FUNCTION_BLOCK StartMovementsTask EXTENDS TcoMitsubishiRoboticsTask
VAR
    _moveParams : TcoAbstractions.TcoRoboticsMovementsParams;
END_VAR

IF Execute() THEN
    IF _progress = 0 THEN
        IF NOT __ISVALIDREF(inoControl) THEN
            _varInfo := __VARINFO(inoControl);
            Messenger.Programming(_sb.Clear().Append('<#Invalid reference: #>').Append(_varInfo.Symbol).ToString()).Pin();
        ELSIF NOT __ISVALIDREF(inoConfig) THEN
            _varInfo := __VARINFO(inoConfig);
            Messenger.Programming(_sb.Clear().Append('<#Invalid reference: #>').Append(_varInfo.Symbol).ToString()).Pin();
        ELSIF NOT __ISVALIDREF(inoStatus) THEN
            _varInfo := __VARINFO(inoStatus);
            Messenger.Programming(_sb.Clear().Append('<#Invalid reference: #>').Append(_varInfo.Symbol).ToString()).Pin();
        ELSE
            _progress := _progress + 1;
        END_IF
    END_IF

    IF _progress = 1 THEN
        _varInfo := __VARINFO(inoStatus.State.OperationEnable);

        THIS^.Messenger.OnCondition(_infoTimer.Q AND NOT inoStatus.State.OperationEnable)
            .Warning(_sb.Clear().Append('<#Waiting for Operation enable! #>').Append(_varInfo.Symbol).ToString());

        _varInfo := __VARINFO(inoStatus.State.AutoEnable);

        THIS^.Messenger.OnCondition(_infoTimer.Q AND NOT inoStatus.State.AutoEnable)
            .Warning(_sb.Clear().Append('<#Waiting for auto enable! #>').Append(_varInfo.Symbol).ToString());

        _varInfo := __VARINFO(inoStatus.State.ServoOn);

        THIS^.Messenger.OnCondition(_infoTimer.Q AND NOT inoStatus.State.ServoOn)
            .Warning(_sb.Clear().Append('<#Waiting for motors are On! #>').Append(_varInfo.Symbol).ToString());

        _varInfo := __VARINFO(inoStatus.State.ErrorReset);

        THIS^.Messenger.OnCondition(_infoTimer.Q AND inoStatus.State.ErrorReset)
            .Warning(_sb.Clear().Append('<#Waiting for system is without errors! #>').Append(_varInfo.Symbol).ToString());

        IF inoStatus.State.OperationEnable AND inoStatus.State.AutoEnable AND inoStatus.State.ServoOn AND NOT inoStatus.State.ErrorReset THEN
            _progress := _progress + 1;
        END_IF
    END_IF;

    IF _progress = 2 THEN
        inoControl.GlobalSpeed := _moveParams.GlobalSpeed;
        inoControl.ToolNo := _moveParams.ToolNo;
        inoControl.WorkobjectNo := _moveParams.WorkobjectNo;
        inoControl.PointNo := _moveParams.PointNo;
        inoControl.UserSpecSpeed1 := _moveParams.UserSpecSpeed1;
        inoControl.UserSpecSpeed2 := _moveParams.UserSpecSpeed2;
        inoControl.Coordinates := _moveParams.Coordinates;
        inoControl.ActionNo := 254;

        IF inoControl.ActionNo = inoStatus.State.ActionNo THEN
            _progress := _progress + 1;
        END_IF
    END_IF;

    IF _progress = 3 THEN
        IF inoStatus.State.GlobalSpeed = _moveParams.GlobalSpeed AND
            inoStatus.State.ToolNo = _moveParams.ToolNo AND
            inoStatus.State.WorkobjectNo = _moveParams.WorkobjectNo AND
            inoStatus.State.PointNo = _moveParams.PointNo AND
            inoStatus.State.UserSpecSpeed1 = _moveParams.UserSpecSpeed1 AND
            inoStatus.State.UserSpecSpeed2 = _moveParams.UserSpecSpeed2 AND
            TcoAbstractions.CoordinatesAreEqual(inoStatus.State.Coordinates,
                _moveParams.Coordinates,
                0.01,
                0.01,
                0.01,
                0.01,
                0.01,
                0.01) THEN
            inoControl.ActionNo := 255;
            _progress := _progress + 1;
        END_IF
    END_IF;

    IF _progress = 4 THEN
        IF inoControl.ActionNo = inoStatus.State.ActionNo THEN
            _progress := _progress + 1;
        END_IF
    END_IF;

    IF _progress = 5 THEN
        Messenger.Info(CONCAT('<#Moving to position ID#>: ', INT_TO_STRING(_moveParams.ActionNo)));
        inoControl.ActionNo := _moveParams.ActionNo;

        IF inoControl.ActionNo = inoStatus.State.ActionNo THEN
            inoControl.ActionNo := 255;
            _progress := _progress + 1;
        END_IF
    END_IF;

    IF _progress = 6 THEN
        IF inoControl.ActionNo = inoStatus.State.ActionNo THEN
            DoneWhen(TRUE);
        END_IF
    END_IF;

    CallTimers(TRUE);
    THIS^.ThrowWhen(_errorTimer.Q OR inoStatus.State.ErrorReset);
END_IF

IF THIS^.Error AND NOT _errorMessage.Pinned THEN
    THIS^.Restore();
END_IF

METHOD PUBLIC FB_init : BOOL
VAR_INPUT
    bInitRetains : BOOL; // if TRUE, the retain variables are initialized (warm start / cold start)
    bInCopyCode : BOOL; // if TRUE, the instance afterwards gets moved into the copy code (online change)
    ParentObject : ITcoObject;
END_VAR
END_METHOD

METHOD INTERNAL InvokeWithParams : ITcoTaskStatus
VAR_INPUT
    inMoveParams : TcoAbstractions.TcoRoboticsMovementsParams;
END_VAR
_moveParams := inMoveParams;
InvokeWithParams := THIS^.Invoke();
END_METHOD

(*~
    <docu>
        <summary>
            Executes when task is aborted.
        </summary>
    </docu>
~*)
METHOD PROTECTED OnAbort
IF __ISVALIDREF(inoStatus) THEN
    THIS^.inoStatus.ActionDescription := '<#Start movements was aborted, while not yet completed!#>';
END_IF;
//inoControl.SoftStop := TRUE;
//inoControl.QuickStop := FALSE;
END_METHOD

(*~
    <docu>
        <summary>
            Executes when task reaches the ```Done``` state .
        </summary>
    </docu>
~*)
METHOD PROTECTED OnDone
IF __ISVALIDREF(inoStatus) THEN
    THIS^.inoStatus.ActionDescription := '<#Start movements finished successfully.#>';
END_IF;

_progress := 0;
END_METHOD

(*~
    <docu>
        <summary>
            Executes when task reaches the ```Error``` state.

        </summary>
    </docu>
~*)
METHOD PROTECTED OnError
VAR
    description : STRING;
END_VAR
description := '<#Start movements finished with error.#>';

IF __ISVALIDREF(inoStatus) THEN
    THIS^.inoStatus.ActionDescription := description;
END_IF;

THIS^._errorMessage.Error(_sb.Clear().Append(description).Append(' To restore acknowledge this alarm.').ToString()).Pin();
END_METHOD

METHOD PROTECTED OnStart
IF __ISVALIDREF(inoStatus) THEN
    THIS^.inoStatus.ActionDescription := '<#Start movements stared.#>';
END_IF;

CallTimers(FALSE);
//inoControl.QuickStop:=FALSE;
//inoControl.SoftStop:=FALSE;
END_METHOD

(*~
    <docu>
        <summary>
            Restores this instance to the Ready state. Can be called explicitly or from within one of the restore mechanisms.
            <para>
                See also <see cref="PlcDocu.TcoCore.TcoTask.AutoRestorable()"/>
            </para>
        </summary>
    </docu>
~*)
METHOD Restore : ITcoRestorable
SUPER^.Restore();
END_METHOD

END_FUNCTION_BLOCK

(* stored: Version 1.1.0.1, ProductVersion 3.1.4024.12
   POU StartMovementsTask: Id {953266c2-376c-05da-069b-8b749a86d7e1}, SpecialFunc None
   Method FB_init: Id {3ab9803b-aeeb-0b6e-3aaf-76c3c2bbfe0c}
   Method InvokeWithParams: Id {ac7bd21c-c9c7-0831-35ca-43103bea2b8b}
   Method OnAbort: Id {190ce994-2dca-0525-2cf5-b44cb0ec880d}
   Method OnDone: Id {bae91270-410e-03a6-32c9-d0949025f448}
   Method OnError: Id {9c2927c7-5b41-0c79-02fd-fcb0df63f5cb}
   Method OnStart: Id {36be574e-cee4-0aef-32b6-999b4cc8718a}
   Method Restore: Id {cbad9b16-e254-04e1-356b-728700ebf737} *)
